// TIA Portal V17 export
// export: Created 2025-06-20T11:55:19.8542396Z, ExportSetting WithDefaults, DisplayName Totally Integrated Automation Portal, DisplayVersion V17 Update 8, DisplayName TIA Portal Openness, DisplayVersion V17 Update 8, DisplayName TIA Portal Version Control Interface, DisplayVersion V17, DisplayName SINAMICS Startdrive Advanced, DisplayVersion V17 SP2, DisplayName SINAMICS Startdrive G110M, G120, G120C, G120D, G120P, G115D, DisplayVersion V17 SP2, DisplayName SINAMICS Startdrive G130, G150, S120, S150, SINAMICS MV, S210, DisplayVersion V17 SP2, DisplayName STEP 7 Professional, DisplayVersion V17 Update 8, DisplayName SINUMERIK ONE STEP 7 Toolbox, DisplayVersion V17 Update 12, DisplayName SINUMERIK ONE PLC Basic Program Plus, DisplayVersion V17 Update 12, DisplayName SINUMERIK 840D sl STEP 7 Toolbox, DisplayVersion V17 Update 12, DisplayName STEP 7 Safety, DisplayVersion V17 Update 6, DisplayName WinCC Advanced, DisplayVersion V17 Update 8
DATA_BLOCK "DB17010_MAINTENANCE_HMI_SCREENS_VARIABLES"   // DB16100
{ S7_Optimized_Access := 'FALSE'; DB_Accessible_From_OPC_UA := 'FALSE' }
VERSION : 0.1
// stored: AutoNumber false, DBAccessibleFromOPCUA false, DBAccessibleFromWebserver true, IsOnlyStoredInLoadMemory false, IsWriteProtectedInAS false
   VAR
      HMI_SIGNALS : Struct
         ACKNOWLEDGE_ACTION_BUTTON : Bool;
         OPERATOR_HELP_VALUE : Int;
         MAINTENANCE_ACTION_LIST_VALUE : Int;
         MAINTENANCE_HMI_VALUE_1 : Int;
         MAINTENANCE_HMI_VALUE_2 : Int;
         MAINTENANCE_HMI_VALUE_3 : Int;
         MAINTENANCE_HMI_VALUE_4 : Int;
         MAINTENANCE_HMI_VALUE_5 : Int;
         MAINTENANCE_HMI_VALUE_6 : Int;
         MAINTENANCE_HMI_VALUE_7 : Int;
         MAINTENANCE_HMI_VALUE_8 : Int;
         MAINTENANCE_HMI_VALUE_9 : Int;
         MAINTENANCE_HMI_VALUE_10 : Int;
         MAINTENANCE_HMI_VALUE_11 : Int;
         MAINTENANCE_HMI_VALUE_12 : Int;
         MAINTENANCE_HMI_BIT_VALUE_1 : Bool;
      END_STRUCT;
   END_VAR
BEGIN
END_DATA_BLOCK
